FUNCTION_BLOCK Calibrate IMPLEMENTS I_CalibrateLinear
VAR
	_Gain	: LREAL := 1;
	_Offset : LREAL := 0;
END_VAR

PROPERTY Gain : LREAL
SET
_Gain := Gain;
END_SET
END_PROPERTY

PROPERTY Offset : LREAL
SET
_Offset := Offset;
END_SET
END_PROPERTY

METHOD Transform : LREAL
VAR_INPUT
	Value	: LREAL;
	Reverse : BOOL := FALSE;
END_VAR
IF Reverse THEN
	Transform := (Value - _Offset) / _Gain;
ELSE
	Transform := Value * _Gain + _Offset;
END_IF
END_METHOD

END_FUNCTION_BLOCK

(* stored: Version 1.1.0.1, ProductVersion 3.1.4026.18
   POU Calibrate: Id {01948038-b423-45e4-b511-93be38eed1bf}, SpecialFunc None
   Property Gain: Id {417c60eb-3c44-47c8-9d43-5599bf08b98d}
   Set Set: Id {c2874b69-f815-4023-b824-20feee542447}
   Property Offset: Id {88bef42c-e99f-4246-8b80-fad72c6ad77d}
   Set Set: Id {e3763bf3-38e4-44a5-a6bf-390e968de54f}
   Method Transform: Id {e24311cc-16f0-41d2-8de5-6f59f19959ff} *)
